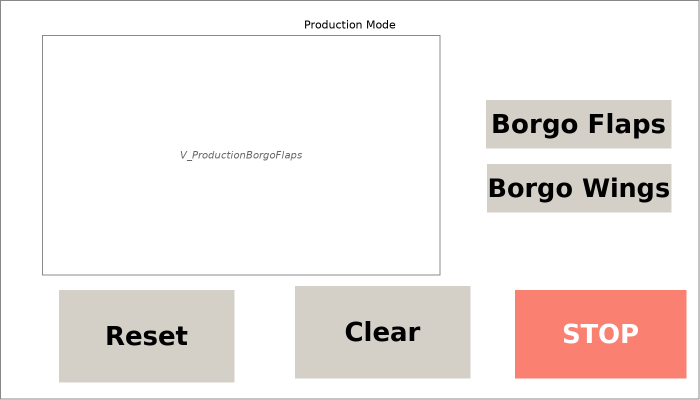
VISUALIZATION V_ProductionModule  // 700x400
VAR_IN_OUT
	HMI : ST_PackMLBaseModule_HMI;
END_VAR
    RoundedRectangle (295,286 175x92), "Clear"
        OnMouseClick: execute { HMI.Command.State := E_PMLCommand.ePMLCommand_Clear; }
    RoundedRectangle (59,290 175x92), "Reset"
        OnMouseClick: execute { HMI.Command.State := E_PMLCommand.ePMLCommand_Reset; }
    RoundedRectangle (513,288 175x92), "STOP"
        toggle GVL_Safety.eStopHMI
        OnMouseClick: execute {  }
    Label (0,0 700x50), "Production Mode"
    Frame (42,35 398x240)
        shows V_ProductionBorgoFlaps()
        shows V_ProductionBorgoWings()
    RoundedRectangle (486,100 185x48), "Borgo Flaps"
        OnMouseClick: execute { HMI.Command.State := E_PMLCommand.ePMLCommand_Clear; }
    RoundedRectangle (487,164 184x48), "Borgo Wings"
        OnMouseClick: execute { HMI.Command.State := E_PMLCommand.ePMLCommand_Clear; }
END_VISUALIZATION

(* stored: Version 1.1.0.1, ProductVersion 3.1.4024.15
   Visu V_ProductionModule: Id {36f6a3ae-b99e-0ef0-3759-f9efb58a3c39} *)
